Staubli VAL3: sendAck.pgx

public program sendAck()
begin
  switch rosGenericMsg.header.nMsgType
    case 11
      call sendTrajPtAck()
    break
    case 14
      call sendTrajPtFAck()
    break
    default
    break
  endSwitch

  // regardless of result from sending ACK
  // reset state machine to receive new messages
  nDataInState=0
end
